{attribute 'qualified_only'}
{attribute 'strict'}
TYPE E_PressureTolerance :
(
	enum_member := 0
);
END_TYPE

(* stored: Version 1.1.0.1, ProductVersion 3.1.4024.12
   DUT E_PressureTolerance: Id {98ab5486-b779-4b8a-b969-233b66211c9d} *)
